TYPE T_ProductDescription : STRING[48];
END_TYPE

(* stored: Version 1.1.0.1, ProductVersion 3.1.4024.15
   DUT T_ProductDescription: Id {0b5d4ad5-e279-41b1-b7cf-82755d9d13b1} *)
